FUNCTION_BLOCK A1
VAR_INPUT
END_VAR
VAR_OUTPUT
END_VAR
VAR
	R1: Recepie1;
	stateReset: INT := 1;
END_VAR

IF stateReset = 0 THEN
	R1();
END_IF

RETURN;

END_FUNCTION_BLOCK

(* stored: Version 1.1.0.1, ProductVersion 3.1.4024.15
   POU A1: Id {8edd17f5-41a6-4587-bf6c-50098ee6fd1d}, SpecialFunc None *)
